INTERFACE ITF_Observer

PROPERTY ID : udint
GET
END_GET
SET
END_SET
END_PROPERTY

METHOD update : BOOL
VAR_INPUT
	Station : REFERENCE TO FB_Station;
END_VAR
END_METHOD

END_INTERFACE

(* stored: Version 1.1.0.1, ProductVersion 3.1.4024.12
   Itf ITF_Observer: Id {5a0a5a3e-cd09-42bf-a75a-19820151c3a1}
   Property ID: Id {629996f4-d3e8-4b77-b1eb-72f9d16b994b}
   Get Get: Id {80963415-adf6-4d17-8e8e-29b3a8537fd7}
   Set Set: Id {c1245ae3-5b0e-439c-95de-620929205529}
   Method update: Id {60239a47-187d-4a1c-ad05-245ee77b08a1} *)
